// TIA Portal project "End Assignment - Alexander Kugelmann" (V17)

(* hardware
DEVICE "HMI_1"  KTP700 Basic PN
   slot 0: "HMI_1"  KTP700 Basic PN  6AV2 123-2GB03-0AX0  17.0.0.0
   slot 1: "HMI_RT_1"  KTP700 Basic PN  6AV2 123-2GB03-0AX0  17.0.0.0
   slot 5: "HMI_1.IE_CP_1"  PROFINET Interface  17.0.0.0
      slot 1: "PROFINET Interface_1"  PROFINET Interface
         slot 1: "Port_1"  Port
DEVICE "S7-1200 station_1"  S7-1200 Station
   slot 0: "Rack_0"  S7-1200 Rack  Rack  V1.0
   slot 1: "PLC_1"  CPU 1215C AC/DC/Rly  6ES7 215-1BG40-0XB0  V4.5
   slot 2: "DI 8x24VDC_1"  6ES7 221-1BF32-0XB0  V2.0
   slot 3: "DQ 8x24VDC _1"  SM 1222 DQ8 x 24VDC  6ES7 222-1BF32-0XB0  V2.0
*)

// ===== PLC "PLC_1"  CPU 1215C AC/DC/Rly =====

VAR_GLOBAL   // PLC tag table "Default tag table"
   "time" AT %MW200 : Int;
   "Clock_Byte" AT %MB0 : Byte;
   "Clock_10Hz" AT %M0.0 : Bool;
   "Clock_5Hz" AT %M0.1 : Bool;
   "Clock_2.5Hz" AT %M0.2 : Bool;
   "Clock_2Hz" AT %M0.3 : Bool;
   "Clock_1.25Hz" AT %M0.4 : Bool;
   "Clock_1Hz" AT %M0.5 : Bool;
   "Clock_0.625Hz" AT %M0.6 : Bool;
   "Clock_0.5Hz" AT %M0.7 : Bool;
   "trigger" AT %M1.0 : Bool;
END_VAR

VAR_GLOBAL   // PLC tag table "Hardware_I_O_Tags"
   "i_DR1_FlowSensorWaste" AT %I0.0 : Bool;
   "i_DR2_FlowSensorProduct" AT %I0.1 : Bool;
   "i_DR3_FlowSensorCocoa" AT %I0.2 : Bool;
   "i_DR4_FlowSensorSugar" AT %I0.3 : Bool;
   "i_RP_Start" AT %I0.4 : Bool;
   "i_RP_CocoaMinus" AT %I0.5 : Bool;
   "i_RP_CocoaPlus" AT %I0.6 : Bool;
   "i_RP_SugarMinus" AT %I0.7 : Bool;
   "i_RP_SugarPlus" AT %I1.0 : Bool;
   "i_RP_AllMilk" AT %I1.1 : Bool;
   "i_CP_CleanMinus" AT %I1.2 : Bool;
   "i_CP_BatchesMinus" AT %I1.3 : Bool;
   "i_CP_BatchesPlus" AT %I1.4 : Bool;
   "i_CP_1Batch" AT %I1.5 : Bool;
   "i_Tank_HeaterFeedback" AT %I8.0 : Bool;
   "i_Tank_LevelLow" AT %I8.1 : Bool;
   "i_Tank_LevelMiddle" AT %I8.2 : Bool;
   "i_Tank_LevelHigh" AT %I8.3 : Bool;
   "i_CP_Start" AT %I8.4 : Bool;
   "o_Tank_ValveWaste" AT %Q0.0 : Bool;
   "o_Tank_ValveProduct" AT %Q0.1 : Bool;
   "o_Tank_ValveCocoa" AT %Q0.2 : Bool;
   "o_Tank_ValveSugar" AT %Q0.3 : Bool;
   "o_Tank_ValveMilk" AT %Q0.4 : Bool;
   "o_Tank_ValveWater" AT %Q0.5 : Bool;
   "o_RP_Started_LED" AT %Q0.6 : Bool;
   "o_RP_Cocoa_LED" AT %Q0.7 : Bool;
   "o_RP_Sugar_LED" AT %Q1.0 : Bool;
   "o_RP_AllMilk_LED" AT %Q1.1 : Bool;
   "o_Tank_LevelEmpty_LED" AT %Q12.0 : Bool;
   "o_Tank_LevelLow_LED" AT %Q12.1 : Bool;
   "o_Tank_LevelMiddle_LED" AT %Q12.2 : Bool;
   "o_Tank_LevelHigh_LED" AT %Q12.3 : Bool;
   "o_Tank_Heater" AT %Q12.4 : Bool;
   "o_Tank_Mixer" AT %Q12.5 : Bool;
   "ai_Tank_Level" AT %IW64 : Int;
   "TankLevelScaledValue" AT %MD0 : Real;
   "ai_Tank_Temperature" AT %IW66 : Int;
   "TankTemperatureScaledValue" AT %MD4 : Real;
END_VAR

DATA_BLOCK "CLock_DB"   // DB1
{ S7_Optimized_Access := 'TRUE' }
VERSION : 0.1
// stored: InstanceOfName CLock
"CLock"
BEGIN
END_DATA_BLOCK

DATA_BLOCK "EM_TankVolume_DB"   // DB3
{ S7_Optimized_Access := 'TRUE' }
VERSION : 0.1
// stored: InstanceOfName EM_TankVolume
"EM_TankVolume"
BEGIN
END_DATA_BLOCK

DATA_BLOCK "EM_TankHeating_DB"   // DB5
{ S7_Optimized_Access := 'TRUE' }
VERSION : 0.1
// stored: InstanceOfName EM_TankHeating
"EM_TankHeating"
BEGIN
END_DATA_BLOCK

DATA_BLOCK "DB_HMI"   // DB7
{ S7_Optimized_Access := 'TRUE' }
VERSION : 0.1
   VAR RETAIN
      start : Bool;
   END_VAR
   VAR
      stop : Bool;
      "tank volume" : Int := 0;
      "volume_level > 0" : Bool;
      "volume_level > 15" : Bool;
      "volume_level > 25" : Bool;
      "volume_level > 50" : Bool;
      "volume_level > 75" : Bool;
      "temperature input" : Int := 50;
      "tank temperature" : Int := 10;
      "add water" : Bool;
      "valve powder" : Bool;
      "booster pump" : Bool;
      "enable heating" : Bool;
      mix : Bool;
      "valve milk" : Bool;
      "milk booster pump" : Bool;
      "valve cocoa" : Bool;
      "valve sugar" : Bool;
   END_VAR
BEGIN
END_DATA_BLOCK

// folder: System blocks/Program resources

DATA_BLOCK "IEC_Counter_0_DB"   // DB2
{ S7_Optimized_Access := 'TRUE' }
AUTHOR : Simatic
FAMILY : IEC
NAME : CNTR
VERSION : 1.0
// stored: InstanceOfName IEC_COUNTER
"IEC_COUNTER"
BEGIN
END_DATA_BLOCK

// folder: Unit_mixerTank/Equipment_01_TankHeating

DATA_BLOCK "CLock_DB_1"   // DB4
{ S7_Optimized_Access := 'TRUE' }
VERSION : 0.1
// stored: InstanceOfName CLock
"CLock"
BEGIN
END_DATA_BLOCK

// folder: (top level)

FUNCTION_BLOCK "CLock"   // FB1, LAD
{ S7_Optimized_Access := 'TRUE' }
VERSION : 0.1
   VAR_INPUT
      trigger : Bool;
      stop : Bool;
   END_VAR
BEGIN

REGION Network 1
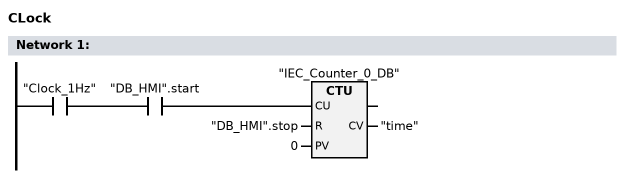
   "IEC_Counter_0_DB".CTU(CU := "Clock_1Hz" AND "DB_HMI".start, R := "DB_HMI".stop, PV := 0, CV => "time");
END_REGION
END_FUNCTION_BLOCK

ORGANIZATION_BLOCK "Main"   // OB1, LAD, ProgramCycle
TITLE = "Main Program Sweep (Cycle)"
{ S7_Optimized_Access := 'TRUE' }
VERSION : 0.1
   VAR_INPUT
      Initial_Call : Bool;   // Initial call of this OB
      Remanence : Bool;   // =True, if remanent data are available
   END_VAR
BEGIN

REGION Network 1
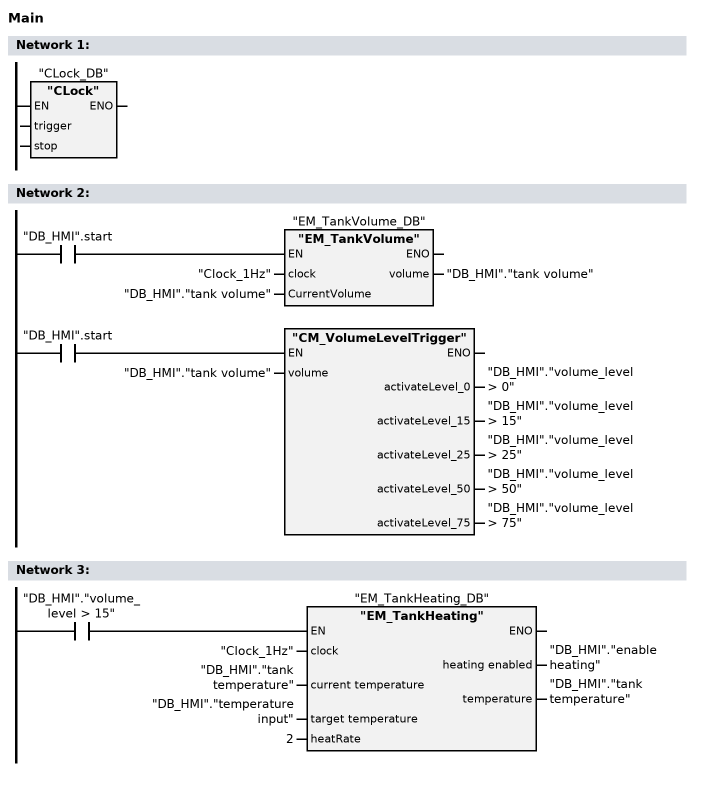
   RUNG wire#powerrail
      "CLock_DB"(trigger :=, stop :=)
   END_RUNG
   // the same network as SCL:
   "CLock_DB"();   // "CLock"
END_REGION

REGION Network 2
   RUNG wire#powerrail
      Contact( "DB_HMI".start )
      "EM_TankVolume_DB"(clock := "Clock_1Hz", CurrentVolume := "DB_HMI"."tank volume", volume => "DB_HMI"."tank volume")
   END_RUNG
   RUNG wire#powerrail
      Contact( "DB_HMI".start )
      "CM_VolumeLevelTrigger"(volume := "DB_HMI"."tank volume", activateLevel_0 => "DB_HMI"."volume_level > 0", activateLevel_15 => "DB_HMI"."volume_level > 15", activateLevel_25 => "DB_HMI"."volume_level > 25", activateLevel_50 => "DB_HMI"."volume_level > 50", activateLevel_75 => "DB_HMI"."volume_level > 75")
   END_RUNG
   // the same network as SCL:
   IF "DB_HMI".start THEN
       "EM_TankVolume_DB"(clock := "Clock_1Hz",   // "EM_TankVolume"
                          CurrentVolume := "DB_HMI"."tank volume",
                          volume => "DB_HMI"."tank volume");
   END_IF;
   IF "DB_HMI".start THEN
       "CM_VolumeLevelTrigger"(volume := "DB_HMI"."tank volume",
                               activateLevel_0 => "DB_HMI"."volume_level > 0",
                               activateLevel_15 => "DB_HMI"."volume_level > 15",
                               activateLevel_25 => "DB_HMI"."volume_level > 25",
                               activateLevel_50 => "DB_HMI"."volume_level > 50",
                               activateLevel_75 => "DB_HMI"."volume_level > 75");
   END_IF;
END_REGION

REGION Network 3
   RUNG wire#powerrail
      Contact( "DB_HMI"."volume_level > 15" )
      "EM_TankHeating_DB"(clock := "Clock_1Hz", "current temperature" := "DB_HMI"."tank temperature", "target temperature" := "DB_HMI"."temperature input", heatRate := 2, "heating enabled" => "DB_HMI"."enable heating", temperature => "DB_HMI"."tank temperature")
   END_RUNG
   // the same network as SCL:
   IF "DB_HMI"."volume_level > 15" THEN
       "EM_TankHeating_DB"(clock := "Clock_1Hz",   // "EM_TankHeating"
                           "current temperature" := "DB_HMI"."tank temperature",
                           "target temperature" := "DB_HMI"."temperature input",
                           heatRate := 2,
                           "heating enabled" => "DB_HMI"."enable heating",
                           temperature => "DB_HMI"."tank temperature");
   END_IF;
END_REGION
END_ORGANIZATION_BLOCK

// folder: Unit_mixerTank/EquipmentModule_00_TankVolume

FUNCTION_BLOCK "EM_TankVolume"   // FB4, LAD
{ S7_Optimized_Access := 'TRUE' }
VERSION : 0.1
   VAR_INPUT
      clock : Bool;
      CurrentVolume : Int;
   END_VAR
   VAR_OUTPUT
      volume : Int;
   END_VAR
   VAR_TEMP
      flowRate : Int;
      trig : Bool;
   END_VAR
BEGIN

REGION Network 1
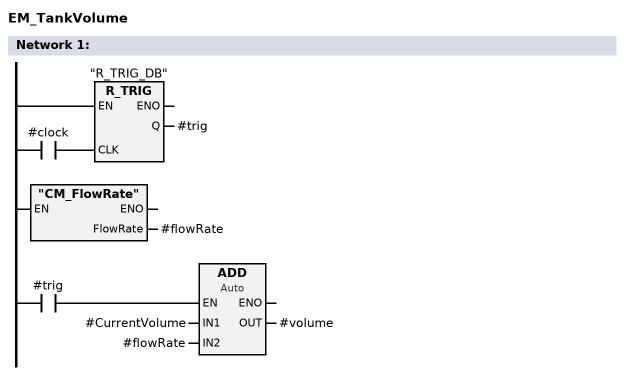
   "R_TRIG_DB"(CLK := #clock, Q => #trig);   // R_TRIG
   "CM_FlowRate"(FlowRate => #flowRate);
   IF #trig THEN #volume := #CurrentVolume + #flowRate; END_IF;
END_REGION
END_FUNCTION_BLOCK

// folder: Unit_mixerTank/EquipmentModule_00_TankVolume/ControlModules

FUNCTION "CM_VolumeLevelTrigger" : Void   // FC1, LAD
{ S7_Optimized_Access := 'TRUE' }
VERSION : 0.1
   VAR_INPUT
      volume : Word;
   END_VAR
   VAR_OUTPUT
      activateLevel_0 : Bool;
      activateLevel_15 : Bool;
      activateLevel_25 : Bool;
      activateLevel_50 : Bool;
      activateLevel_75 : Bool;
   END_VAR
BEGIN

REGION Network 1
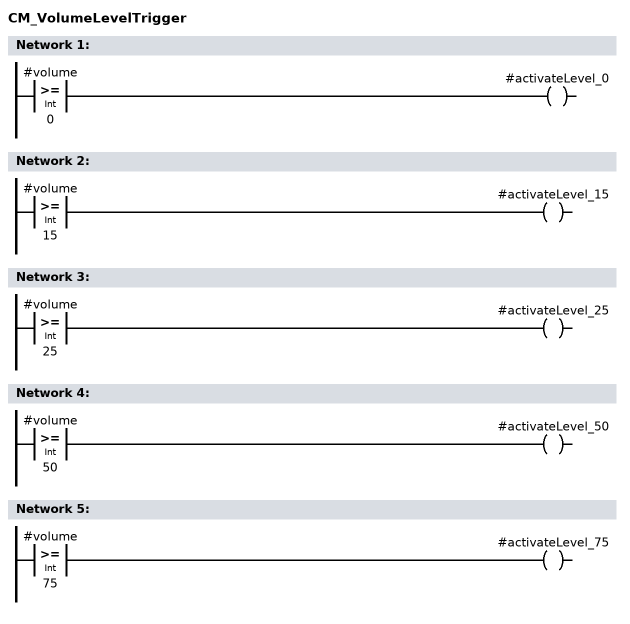
   RUNG wire#powerrail
      { S7_Templates := "SrcType := Int" } GE_Contact(in1 := #volume, in2 := 0)
      Coil( #activateLevel_0 )
   END_RUNG
   // the same network as SCL:
   #activateLevel_0 := #volume >= 0;
END_REGION

REGION Network 2
   RUNG wire#powerrail
      { S7_Templates := "SrcType := Int" } GE_Contact(in1 := #volume, in2 := 15)
      Coil( #activateLevel_15 )
   END_RUNG
   // the same network as SCL:
   #activateLevel_15 := #volume >= 15;
END_REGION

REGION Network 3
   RUNG wire#powerrail
      { S7_Templates := "SrcType := Int" } GE_Contact(in1 := #volume, in2 := 25)
      Coil( #activateLevel_25 )
   END_RUNG
   // the same network as SCL:
   #activateLevel_25 := #volume >= 25;
END_REGION

REGION Network 4
   RUNG wire#powerrail
      { S7_Templates := "SrcType := Int" } GE_Contact(in1 := #volume, in2 := 50)
      Coil( #activateLevel_50 )
   END_RUNG
   // the same network as SCL:
   #activateLevel_50 := #volume >= 50;
END_REGION

REGION Network 5
   RUNG wire#powerrail
      { S7_Templates := "SrcType := Int" } GE_Contact(in1 := #volume, in2 := 75)
      Coil( #activateLevel_75 )
   END_RUNG
   // the same network as SCL:
   #activateLevel_75 := #volume >= 75;
END_REGION
END_FUNCTION

FUNCTION "CM_VolumeSensor" : Void   // FC3, LAD
TITLE = Read the volume sensor
{ S7_Optimized_Access := 'TRUE' }
VERSION : 0.1
// A fysical analog input is connected with a sensor what measures the height of the fluid level in the tank
   VAR_INPUT
      CurrentVolume : Int;
   END_VAR
   VAR_OUTPUT
      VolumePercentage : Real;
   END_VAR
   VAR_TEMP
      NormValueVolumeInput : Real;
   END_VAR
   VAR CONSTANT
      "tank volume" : Int := 100;
   END_VAR
BEGIN

REGION Network 1: Read analog input
   // Normalize analog input -> norm value (0.0 - 1.0)
   // Scale value to read the volume of a tank,
   // => scaling out a value for the tank is normalized from a volume of 0.0 (empty) to 100.0 procent (full).
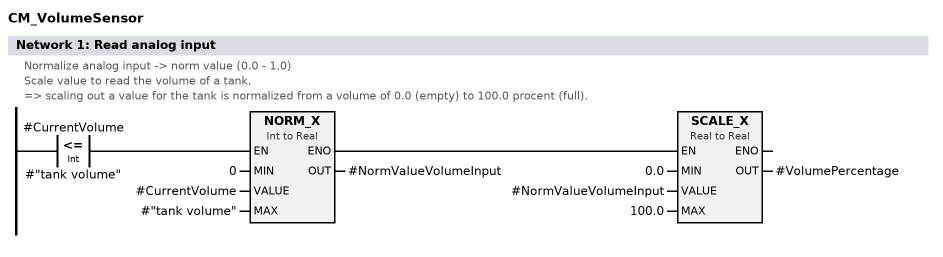
   RUNG wire#powerrail
      { S7_Templates := "SrcType := Int" } LE_Contact(in1 := #CurrentVolume, in2 := #"tank volume")
      { S7_Templates := "[SrcType := Int, DestType := Real]" } Normalize(min := 0, value := #CurrentVolume, max := #"tank volume", out => #NormValueVolumeInput)
      { S7_Templates := "[SrcType := Real, DestType := Real]" } Scale(min := 0.0, value := #NormValueVolumeInput, max := 100.0, out => #VolumePercentage)
   END_RUNG
   // the same network as SCL:
   IF #CurrentVolume <= #"tank volume" THEN
       #NormValueVolumeInput := NORM_X(MIN := 0, VALUE := #CurrentVolume, MAX := #"tank volume");
       #VolumePercentage := SCALE_X(MIN := 0.0, VALUE := #NormValueVolumeInput, MAX := 100.0);
   END_IF;
END_REGION
END_FUNCTION

FUNCTION "CM_FlowRate" : Void   // FC5, LAD
{ S7_Optimized_Access := 'TRUE' }
VERSION : 0.1
   VAR_OUTPUT
      FlowRate : Int;
   END_VAR
   VAR_TEMP
      trig : Bool;
   END_VAR
BEGIN

REGION Network 1
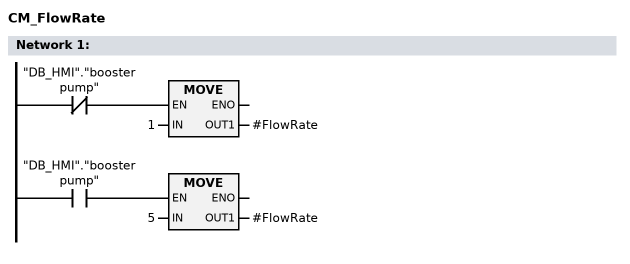
   RUNG wire#powerrail
      I_Contact( "DB_HMI"."booster pump" )
      Move(in := 1, out1 => #FlowRate)
   END_RUNG
   RUNG wire#powerrail
      Contact( "DB_HMI"."booster pump" )
      Move(in := 5, out1 => #FlowRate)
   END_RUNG
   // the same network as SCL:
   IF NOT "DB_HMI"."booster pump" THEN #FlowRate := 1; END_IF;
   IF "DB_HMI"."booster pump" THEN #FlowRate := 5; END_IF;
END_REGION
END_FUNCTION

// folder: Unit_mixerTank/Equipment_01_TankHeating

FUNCTION_BLOCK "EM_TankHeating"   // FB2, LAD
{ S7_Optimized_Access := 'TRUE' }
VERSION : 0.1
   VAR_INPUT
      clock : Bool;
      "current temperature" : Int;
      "target temperature" : Int;
      heatRate : Int;
   END_VAR
   VAR_OUTPUT
      "heating enabled" : Bool;
      temperature : Int;
   END_VAR
   VAR_TEMP
      trig : Bool;
   END_VAR
   VAR_TEMP   // added for the SCL form of the ladder/FBD networks
      _w1 : Bool;
   END_VAR
BEGIN

REGION Network 1
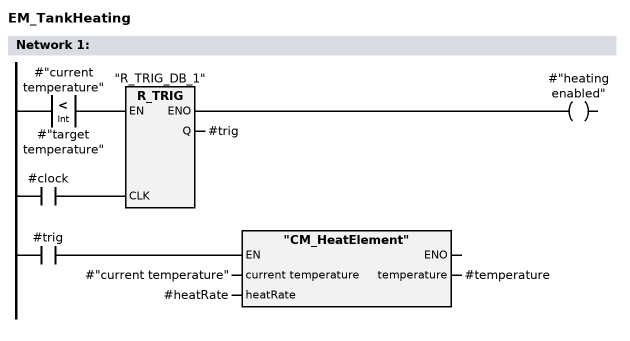
   // ENO of a box is taken as its EN; it also drops when the box reports an error
   #_w1 := #"current temperature" < #"target temperature";
   IF #_w1 THEN
       "R_TRIG_DB_1"(CLK := #clock, Q => #trig);   // R_TRIG
   END_IF;
   #"heating enabled" := #_w1;
   IF #trig THEN
       "CM_HeatElement"("current temperature" := #"current temperature",
                        heatRate := #heatRate,
                        temperature => #temperature);
   END_IF;
END_REGION
END_FUNCTION_BLOCK

// folder: Unit_mixerTank/Equipment_01_TankHeating/ControlModules

FUNCTION "CM_HeatElement" : Void   // FC2, LAD
{ S7_Optimized_Access := 'TRUE' }
VERSION : 0.1
   VAR_INPUT
      "current temperature" : Int;
      heatRate : Int;
   END_VAR
   VAR_OUTPUT
      temperature : Int;
   END_VAR
BEGIN

REGION Network 1
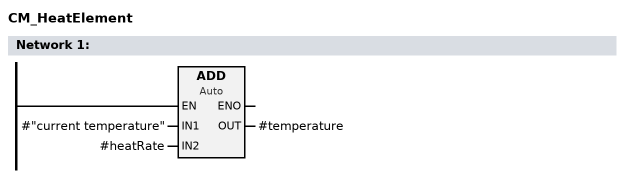
   RUNG wire#powerrail
      Add(in1 := #"current temperature", in2 := #heatRate, out => #temperature)
   END_RUNG
   // the same network as SCL:
   #temperature := #"current temperature" + #heatRate;
END_REGION
END_FUNCTION

// folder: Unit_mixerTank/Equipment_10_FluidInput

FUNCTION_BLOCK "Block_1"   // FB3, LAD
{ S7_Optimized_Access := 'TRUE' }
VERSION : 0.1
BEGIN
END_FUNCTION_BLOCK

(* ===== HMI "HMI_RT_1" =====
system functions are stored by id; their names below are inferred from use
connection "HMI_Connection_1": ETHERNET, SMART_S7_1200_OMS

HMI tags "Default tag table"
   "Tag_ScreenNumber" : UInt, internal
   "DB_HMI_start" : Bool = PLC DB_HMI.start, 1 s
   "DB_HMI_tank volume" : Int = PLC DB_HMI."tank volume", 1 s
   "DB_HMI_tank temperature" : Int = PLC DB_HMI."tank temperature", 1 s
   "time" : Int = PLC time AT %MW200, 1 s
   "DB_HMI_temperature input" : Int = PLC DB_HMI."temperature input", 1 s
   "DB_HMI_enable heating" : Bool = PLC DB_HMI."enable heating", 1 s
   "DB_HMI_stop" : Bool = PLC DB_HMI.stop, 1 s
   "ai_Tank_Temperature" : Int = PLC ai_Tank_Temperature AT %IW66, 1 s
   "DB_HMI_volume_level > 25" : Bool = PLC DB_HMI."volume_level > 25", 1 s
   "DB_HMI_volume_level > 50" : Bool = PLC DB_HMI."volume_level > 50", 1 s
   "DB_HMI_volume_level > 75" : Bool = PLC DB_HMI."volume_level > 75", 1 s
   "DB_HMI_booster pump" : Bool = PLC DB_HMI."booster pump", 1 s

text list "Text_list_1": 0..100 ''

Template "Template_1" 800x480
   Button "Exit" at 714,429 size 71x50; TextOff 'Exit'; PictureOff "ExitRuntime_KTP700_Basic_PN_TR"; PictureOn "ExitRuntime_KTP700_Basic_PN_TR"
      on Release: StopRuntime(0)
   Button "Template_Button" at 614,429 size 71x50; TextOff 'Text'
   Button "Template_Button_1" at 514,429 size 71x50; TextOff 'Text'
   Button "Template_Button_2" at 414,429 size 71x50; TextOff 'Text'
   Button "Template_Button_3" at 314,429 size 71x50; TextOff 'Text'
   Button "Template_Button_4" at 214,429 size 71x50; TextOff 'Text'
   Button "Alarms" at 114,429 size 71x50; TextOff 'Alarms'; PictureOff "AlarmDisplay_KTP700_Basic_PN_TR"; PictureOn "AlarmDisplay_KTP700_Basic_PN_TR"
      on Release: function_ef3f5d25("Alarm window_Unacknowledged", -1)
   Button "Start screen" at 14,429 size 71x50; TextOff 'Start screen'; PictureOff "NavigateHome_KTP700_Basic_PN_TR"; PictureOn "NavigateHome_KTP700_Basic_PN_TR"
      on Release: ActivateScreen("screen_mixerTank", 0)
   SymbolicIOField "Symbolic_IO_Field_Screen" at 93,9 size 600x33; TextOff '0'; TextOn '1'; TextList "TextList_ScreenNames"
      ProcessValue <- "Tag_ScreenNumber"
      on Change: ActivateScreenByNumber("Tag_ScreenNumber", 0)
   DateTimeField "HmiScreenItemData" at 695,25 size 105x25
   DateTimeField "HmiScreenItemData_1" at 695,0 size 105x25
   GraphicView "Logo" at 0,0 size 91x51; Picture "Logo of HMI_1"

screen "screen_mixerTank" 800x480, template "Template_1"
   on GenerateScreen: SetTag("Tag_ScreenNumber", 1)
   TextField "Text field_3" at 634,115 size 51x23; Text 'TANK'
   GraphicView "Graphic view_1" at 527,138 size 269x285; Picture "Graphic_18"
   Button "HmiScreenItemData" at 8,64 size 120x47; TextOff 'HOME'; TextOn 'Screen0'; PictureOff "Navigates to Screen0 for KTP700 Basic+ PN 17.0.0.0"; PictureOn "Navigates to Screen0 for KTP700 Basic+ PN 17.0.0.0"
      on Release: ActivateScreen("screen_home", 0)
   Button "Button_2" at 9,303 size 130x109; TextOff 'EMERGENCY STOP'
      on Press: SetBit("DB_HMI_stop"); ResetBit("DB_HMI_start")
   Button "Button_1" at 7,138 size 128x52; TextOff 'START/PAUSE'
      on Press: InvertBit("DB_HMI_start"); ResetBit("DB_HMI_stop")
   TextField "Text field_5" at 345,23 size 110x23; Text 'MIXER TANK'
   IOField "I/O field_1" at 622,19 size 66x30; FormatPattern s99999
      ProcessValue <- "time"
   TextField "Text field_6" at 528,26 size 84x15; Text 'TIME ELAPSED:'
   TextField "Text field_7" at 473,181 size 45x17; Text 'WATER'
   TextField "Text field_8" at 458,146 size 68x23; Text 'VALVES'
   GraphicIOField "PlotLight_Round_R_1" at 542,180 size 31x31; PictureOn "PilotLight_Round_R_On_256c"; PictureOff "PilotLight_Round_R_Off_256c"
      ProcessValue <- "DB_HMI_volume_level > 25"
   TextField "Text field_9" at 473,265 size 44x17; Text 'SUGAR'
   GraphicIOField "PlotLight_Round_R_2" at 542,267 size 31x31; PictureOff "PilotLight_Round_R_Off_256c"; PictureOn "PilotLight_Round_R_On_256c"
      ProcessValue <- "DB_HMI_volume_level > 50"
   TextField "Text field_10" at 472,307 size 43x17; Text 'COCOA'
   GraphicIOField "PlotLight_Round_R_3" at 542,306 size 31x31; PictureOff "PilotLight_Round_R_Off_256c"; PictureOn "PilotLight_Round_R_On_256c"
      ProcessValue <- "DB_HMI_volume_level > 75"
   TextField "Text field_2" at 154,81 size 145x18; Text 'TARGET TEMPERATURE'
   GraphicIOField "PlotLight_Round_R_4" at 703,345 size 31x31; PictureOff "PilotLight_Round_R_Off_256c"; PictureOn "PilotLight_Round_R_On_256c"
      ProcessValue <- "DB_HMI_enable heating"
   TextField "Text field_11" at 597,348 size 91x20; Text 'Heat Element'
   Bar "Bar_1" at 644,176 size 136x163; MinimumValue 0; MaximumValue 100
      ProcessValue <- "DB_HMI_tank volume"
   TextField "Text field_1" at 688,149 size 37x23; Text 'VOL'
   Bar "Bar_2" at 606,176 size 37x162; MinimumValue 0; MaximumValue 80
      ProcessValue <- "DB_HMI_tank temperature"
   TextField "Text field_4" at 598,149 size 51x23; Text 'TEMP'
   IOField "I/O field_2" at 306,74 size 51x31; FormatPattern s99999
      ProcessValue <- "DB_HMI_temperature input"
   TextField "Text field_12" at 472,222 size 33x17; Text 'MILK'
   GraphicIOField "PlotLight_Round_R_5" at 542,222 size 31x31; PictureOff "PilotLight_Round_R_Off_256c"; PictureOn "PilotLight_Round_R_On_256c"
      ProcessValue <- "DB_HMI_volume_level > 25"
   Group "Group" at 631,115 size 62x23
   GraphicIOField "PlotLight_Square_R" at 552,77 size 60x19; PictureOn "PilotLight_Square_R_On_256c"; PictureOff "PilotLight_Square_R_Off_256c"
      ProcessValue <- "DB_HMI_stop"
   GraphicIOField "PlotLight_Square_G" at 552,95 size 60x18; PictureOn "PilotLight_Square_G_On_256c"; PictureOff "PilotLight_Square_G_Off_256c"
      ProcessValue <- "DB_HMI_start"
   Button "Button_4" at 153,376 size 162x36; TextOff 'TOGGLE BOOSTER PUMP'
      on Press: InvertBit("DB_HMI_booster pump")
   GraphicIOField "PlotLight_Round_R" at 322,376 size 36x35; PictureOn "PilotLight_Round_R_On_256c"; PictureOff "PilotLight_Round_R_Off_256c"
      ProcessValue <- "DB_HMI_booster pump"

screen "screen_bottleConveyor" 800x480, template "Template_1"
   on GenerateScreen: SetTag("Tag_ScreenNumber", 2)
   TextField "Text field_5" at 316,14 size 165x23; Text 'BOTTLE CONVEYOR'
   Button "HmiScreenItemData" at 8,64 size 120x47; TextOn 'Screen0'; TextOff 'HOME'; PictureOn "Navigates to Screen0 for KTP700 Basic+ PN 17.0.0.0"; PictureOff "Navigates to Screen0 for KTP700 Basic+ PN 17.0.0.0"
      on Release: ActivateScreen("screen_home", 0)

screen "screen_home" 800x480
   Button "Button_1" at 107,131 size 170x69; TextOff 'MIXER TANK'
      on Release: ActivateScreen("screen_mixerTank", 1)
   Button "Button_2" at 313,131 size 180x68; TextOff 'BOTTLE CONVEYOR'
      on Release: ActivateScreen("screen_bottleConveyor", 2)
   Button "Button_3" at 536,132 size 174x68; TextOff 'SYSTEM OVERVIEW'
      on Release: ActivateScreen("screen_systemOverview", 3)
   Button "Button_4" at 107,319 size 170x69; TextOff 'START PROCESS'
      on Release: ActivateScreen("screen_mixerTank", 1)
   Button "Button_5" at 536,319 size 170x69; TextOff 'STOP PROCESS'
      on Release: ActivateScreen("screen_mixerTank", 1)
   TextField "Text field_5" at 367,14 size 53x23; Text 'HOME'

screen "screen_systemOverview" 800x480
   TextField "Text field_5" at 316,14 size 165x23; Text 'SYSTEM OVERVIEW'
   Button "HmiScreenItemData" at 8,64 size 120x47; TextOn 'Screen0'; TextOff 'HOME'; PictureOn "Navigates to Screen0 for KTP700 Basic+ PN 17.0.0.0"; PictureOff "Navigates to Screen0 for KTP700 Basic+ PN 17.0.0.0"
      on Release: ActivateScreen("screen_home", 0)
*)